FUNCTION_BLOCK RS (* IEC 61131-3 Table 34,#2 *)
  (* Standard: 61131-3 *)
  (* Version 0.0, 2004-12-15, JHC, Rockwell Automation, Converted from SRC format. *)
  (* Compiler header: package fb.rt.plc; *)
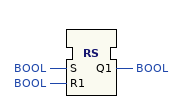
  VAR_INPUT
    S : BOOL;
    R1 : BOOL;
  END_VAR
  VAR_OUTPUT
    Q1 : BOOL;
  END_VAR
  ALGORITHM REQ IN ST:
IF R1 THEN Q1:=false;
ELSIF S THEN Q1:=TRUE;
END_IF;
  END_ALGORITHM
END_FUNCTION_BLOCK
